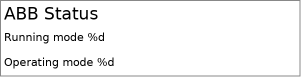
VISUALIZATION _VisuABBStatus  // 301x77
    Label (1,1 148x25), "ABB Status"
    Rectangle (1,25 298x25), "Running mode %d", text variable: ComGVL._gABBRunTable[ComGVL._fbTryOutABBRunMode ]
    Rectangle (1,50 298x25), "Operating mode %d", text variable: ComGVL._gABBOpTable[ComGVL._fbTryOutABBOpMode ]
END_VISUALIZATION

(* stored: Version 1.1.0.1, ProductVersion 3.1.4024.2
   Visu _VisuABBStatus: Id {4883d084-aa3c-48f1-b7e9-b0e91e01458f} *)
